// Mitsubishi GX Works2 project: exa   PLC: FX1N/FX1NC

PROGRAM MAIN
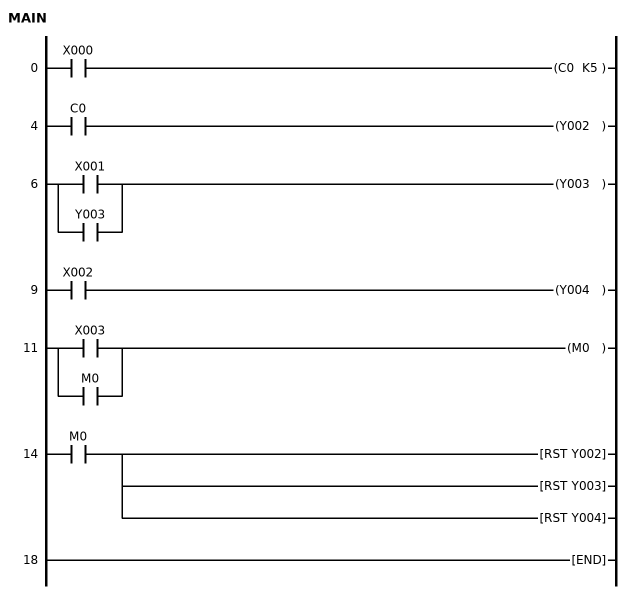
0     LD      X000
      OUT     C0 K5
4     LD      C0
      OUT     Y002
6     LD      X001
      OR      Y003
      OUT     Y003
9     LD      X002
      OUT     Y004
11    LD      X003
      OR      M0
      OUT     M0
14    LD      M0
      RST     Y002
      RST     Y003
      RST     Y004
18    END
END_PROGRAM
